FUNCTION_BLOCK Motor_VS_HMI (* Service Interface Function Block Type *)
  (* Standard: 61499-2 *)
  (* Version 0.0, 6/2/2026, Schneider Electric, template *)
  PACKAGE SE.Nereda;
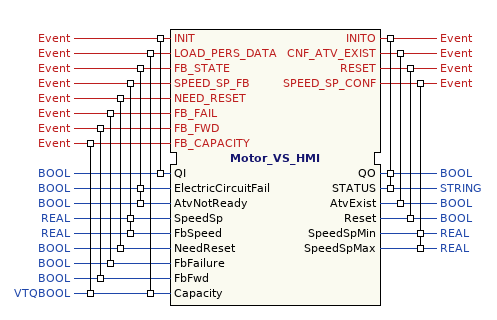
  EVENT_INPUT
    INIT WITH QI;
    LOAD_PERS_DATA WITH Capacity;
    FB_STATE WITH ElectricCircuitFail, AtvNotReady;
    SPEED_SP_FB WITH SpeedSp, FbSpeed;
    NEED_RESET WITH NeedReset;
    FB_FAIL WITH FbFailure;
    FB_FWD WITH FbFwd;
    FB_CAPACITY WITH Capacity;
  END_EVENT
  EVENT_OUTPUT
    INITO WITH QO, STATUS;
    CNF_ATV_EXIST WITH AtvExist;
    RESET WITH Reset;
    SPEED_SP_CONF WITH SpeedSpMin, SpeedSpMax;
  END_EVENT
  VAR_INPUT
    QI : BOOL;
    ElectricCircuitFail : BOOL;
    AtvNotReady : BOOL;
    SpeedSp : REAL;
    FbSpeed : REAL;
    NeedReset : BOOL;
    FbFailure : BOOL;
    FbFwd : BOOL; (* Status Run *)
    Capacity : VTQBOOL;
  END_VAR
  VAR_OUTPUT
    QO : BOOL; (* Event Output Qualifier *)
    STATUS : STRING; (* Service Status *)
    AtvExist : BOOL;
    Reset : BOOL;
    SpeedSpMin : REAL;
    SpeedSpMax : REAL;
  END_VAR
  SERVICE /
    SEQUENCE 
    END_SEQUENCE
  END_SERVICE
END_FUNCTION_BLOCK
